TYPE Heater :
STRUCT
	Setpoint : INT;
	Alarm : BOOL;
	Name : STRING;
	Current : REAL;
END_STRUCT
END_TYPE

(* stored: Version 1.1.0.1, ProductVersion 3.1.4024.12
   DUT Heater: Id {33757206-8621-4a8d-b835-9a6a088a3b24} *)
